FUNCTION_BLOCK CROSSCOMM_SENDER_160EC6DC30B01CA3B (* Service Interface Function Block Type *)
  (* Standard: 61499-2 *)
  (* Version 0.0, 9/22/2017, bababen, nxtControl GmbH, template *)
  PACKAGE Main;
  (* Compiler Cpp nxtControl builtin 1.0 *)
  {SET_ATTRIBUTE(Runtime.FBType.ImplementingType, Runtime.System#DYNGEN_CROSSCOMM_SENDER)}
  {SET_ATTRIBUTE(Configuration.GenericFBType.InterfaceParams, Runtime.System#<InterfaceList> <EventInputs> <Event Name="INITO"> <With Var="PushRetracted" /> <With Var="PushExtended" /> <With Var="LuggageArrived" /> <With Var="LuggageLifted" /> </Event> <Event Name="CNF"> <With Var="PushRetracted" /> <With Var="PushExtended" /> <With Var="LuggageArrived" /> <With Var="LuggageLifted" /> </Event> </EventInputs> <InputVars> <VarDeclaration Name="PushRetracted" Type="BOOL" /> <VarDeclaration Name="PushExtended" Type="BOOL" /> <VarDeclaration Name="LuggageArrived" Type="BOOL" /> <VarDeclaration Name="LuggageLifted" Type="BOOL" /> </InputVars> </InterfaceList>)}
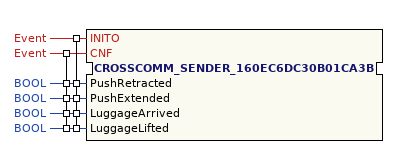
  EVENT_INPUT
    INITO WITH PushRetracted, PushExtended, LuggageArrived, LuggageLifted;
    CNF WITH PushRetracted, PushExtended, LuggageArrived, LuggageLifted;
  END_EVENT
  VAR_INPUT
    PushRetracted : BOOL;
    PushExtended : BOOL;
    LuggageArrived : BOOL;
    LuggageLifted : BOOL;
  END_VAR
  EC_STATES
    START;
  END_STATES
END_FUNCTION_BLOCK
